VAR_GLOBAL CONSTANT
	nMaxStationCount : UINT := 10; // Used To Size StationConfig Arrays
END_VAR
VAR_GLOBAL
	nNumOfActiveStation	: UINT := 1; // Default min one station exist
END_VAR

(* stored: Version 1.1.0.1
   GVL GVL_StationConfig: Id {dca36831-11de-0605-3b71-366dc1955369} *)
